{attribute 'GeneratedUsingTerminal: AES-D-BC-ECAT Gen2-0001'}
{attribute addProperty BoxType "AES-D-BC-ECAT Gen2-0001"}
{attribute addProperty Id "digital_Data_IAT %I*ARRAY[0..31] OF USINT32"}
{attribute addProperty CRC "1374483313"}
{attribute addProperty Size "32"}
TYPE Inputs_23559BB0 EXTENDS TcoIo.InputBase_8311D824 :
STRUCT
	{attribute addProperty Name "digital_Data_I"}
	digital_Data_I AT %I* : ARRAY[0..31] OF USINT;
END_STRUCT
END_TYPE

(* stored: Version 1.2.0.0
   DUT Inputs_23559BB0: Id {dbebdb8b-1877-40cd-a947-c8f511b77b75} *)
